{attribute 'GeneratedUsingTerminal: EK1100-0000-0018'}
{attribute addProperty BoxType "EK1100-0000-0018"}
{attribute addProperty Id "Term_232_EL1809EL1809_32157CFD20"}
{attribute addProperty CRC "1875807467"}
{attribute addProperty Size "20"}
{attribute addProperty Name "Term 231 (EK1100)"}
TYPE Term_231_EK1100_6FCE8CEB EXTENDS EK1100_1FC0878B :
STRUCT
	{attribute addProperty Name "Term 232 (EL1809)"}
	{attribute addProperty PreviousPort "Term 231 (EK1100) : B"}
	{attribute addProperty SyncUnit "default"}
	Term_232_EL1809 : EL1809_32157CFD;
END_STRUCT
END_TYPE

(* stored: Version 1.2.0.0, ProductVersion 3.1.4024.11
   DUT Term_231_EK1100_6FCE8CEB: Id {ebd4f6e3-345a-4510-b695-9711b53d5572} *)
